FUNCTION_BLOCK FB_Grundablauf EXTENDS FB_Basis
VAR_INPUT
	// Instanzieren von Reaktor mit Interface
	Reaktor			:I_Reaktor;
	
	// Prozessparameter
	SekReakt		:INT;
	Temp			:REAL;
	Entleermenge	:REAL;
	Pumpmenge		:REAL;
	Haltedauer		:INT;
	Ruehrdauer		:INT;
	Wartedauer		:INT;
	Zirkulierdauer	:INT;
END_VAR
VAR_OUTPUT
	CW				:RezeptControlWord;
END_VAR
VAR
	Leitung			:INT := 1;
	LeitungsCheck	:BOOL := TRUE;
END_VAR

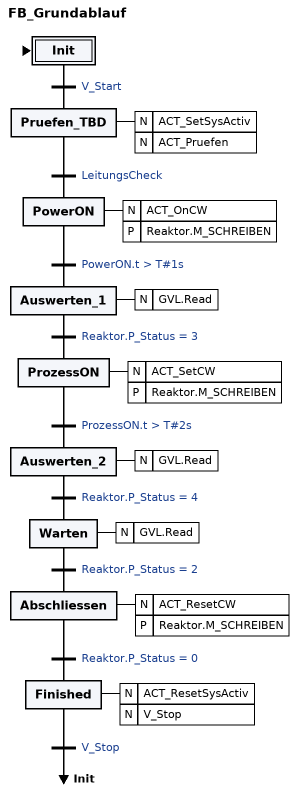
INITIAL_STEP Init:
END_STEP
TRANSITION FROM Init TO Pruefen_TBD
    := V_Start;
END_TRANSITION
STEP Pruefen_TBD:
    ACT_SetSysActiv(N);
    ACT_Pruefen(N);
END_STEP
TRANSITION FROM Pruefen_TBD TO PowerON
    := LeitungsCheck;
END_TRANSITION
STEP PowerON:
    ACT_OnCW(N);
    Reaktor.M_SCHREIBEN(P);
END_STEP
TRANSITION FROM PowerON TO Auswerten_1
    := PowerON.t > T#1s;
END_TRANSITION
STEP Auswerten_1:
    GVL.Read(N);
END_STEP
TRANSITION FROM Auswerten_1 TO ProzessON
    := Reaktor.P_Status = 3;
END_TRANSITION
STEP ProzessON:
    ACT_SetCW(N);
    Reaktor.M_SCHREIBEN(P);
END_STEP
TRANSITION FROM ProzessON TO Auswerten_2
    := ProzessON.t > T#2s;
END_TRANSITION
STEP Auswerten_2:
    GVL.Read(N);
END_STEP
TRANSITION FROM Auswerten_2 TO Warten
    := Reaktor.P_Status = 4;
END_TRANSITION
STEP Warten:
    GVL.Read(N);
END_STEP
TRANSITION FROM Warten TO Abschliessen
    := Reaktor.P_Status = 2;
END_TRANSITION
STEP Abschliessen:
    ACT_ResetCW(N);
    Reaktor.M_SCHREIBEN(P);
END_STEP
TRANSITION FROM Abschliessen TO Finished
    := Reaktor.P_Status = 0;
END_TRANSITION
STEP Finished:
    ACT_ResetSysActiv(N);
    V_Stop(N);
END_STEP
TRANSITION FROM Finished TO Init
    := V_Stop;
END_TRANSITION

ACTION ACT_OnCW:
CW.PowerOn := TRUE;
END_ACTION

ACTION ACT_Pruefen:
// TBD
END_ACTION

ACTION ACT_ResetCW:
CW.PowerOn := FALSE;
CW.SekReakt := 0;
CW.Leitung := 0;
CW.Temp := 0;
CW.Enlteermenge := 0;
CW.Pumpmenge := 0;
CW.Haltedauer := 0;
CW.Ruehrdauer := 0;
CW.Wartedauer := 0;
CW.Zirkulierdauer := 0;
END_ACTION

ACTION ACT_ResetSysActiv:
GVL.SysState := 1;
END_ACTION

ACTION ACT_SetCW:
CW.SekReakt := SekReakt;
CW.Leitung := Leitung;
CW.Temp := Temp;
CW.Enlteermenge := Entleermenge;
CW.Pumpmenge := Pumpmenge;
CW.Haltedauer := Haltedauer;
CW.Ruehrdauer := Ruehrdauer;
CW.Wartedauer := Wartedauer;
CW.Zirkulierdauer := Zirkulierdauer;
END_ACTION

ACTION ACT_SetSysActiv:
GVL.SysState := 2;
END_ACTION

END_FUNCTION_BLOCK

(* stored: Version 1.1.0.1, ProductVersion 3.1.4024.12
   POU FB_Grundablauf: Id {ba376277-9321-4613-a760-dc59dad2be70}, SpecialFunc None
   Action ACT_OnCW: Id {bbfb5b7b-4199-42ab-9867-4383501d60cb}
   Action ACT_Pruefen: Id {0cd24355-6c1e-4b69-9cae-0f7a68be8849}
   Action ACT_ResetCW: Id {3b8b9e9b-9340-4e2a-be39-cdb306c65fb9}
   Action ACT_ResetSysActiv: Id {7cf457ea-1d08-461d-a894-7e22b2ced456}
   Action ACT_SetCW: Id {3463accb-09f1-4209-8b67-a7a4a1be2267}
   Action ACT_SetSysActiv: Id {efdd272f-178e-49f6-986a-deaf9af92096} *)
